// TwinCAT 3 PLC project PLC
// ProgramVersion: 3.1.4023.0
// libraries:
//   Tc2_Standard, * (Beckhoff Automation GmbH)
//   Tc2_System, * (Beckhoff Automation GmbH)
//   Tc2_Utilities, * (Beckhoff Automation GmbH)
//   Tc3_Module, * (Beckhoff Automation GmbH)
//   Util, * (System)
// project tree:
//   / PlcTask.TcTTO
//   POUs/ FB_ExportScopeData.TcPOU, FB_ScopeServerSample.TcPOU, MAIN.TcPOU
// real-time tasks:
//   TASK PlcTask: cycle T#10ms, priority 20, ADS port 350

CONFIGURATION PLC
    RESOURCE PLC ON TwinCAT3
        TASK PlcTask(INTERVAL := T#10ms, PRIORITY := 20);
        PROGRAM MAIN WITH PlcTask : MAIN;
    END_RESOURCE
END_CONFIGURATION

// ---- POUs/MAIN.TcPOU
PROGRAM MAIN
VAR
	fbBlink				:BLINK;
	Sinus				:GEN;
	SawTooth			:GEN;
	
	
	fbScopeServer		:FB_ScopeServerSample;
	
	xStartStopScope		:BOOL;
	xScopeBusy			:BOOL;
	xScopeError			:BOOL;
	iScopeErrorID		:UDINT;
	
	
	fbExportToCSV		:FB_ExportScopeData;
	xExport				:BOOL;
	xExportBusy			:BOOL;
	xExportError		:BOOL;
	iExportErrorID		:UDINT;
	
	
	//Example for listing files in a direcorty 
	//https://infosys.beckhoff.com/content/1033/tcplclib_tc2_utilities/35410571.html?id=3151343736833681439	
END_VAR

fbBlink(ENABLE:=TRUE , TIMELOW:=T#200MS , TIMEHIGH:=T#400MS);
Sinus(MODE:=GEN_MODE.SINUS , BASE:=TRUE , PERIOD:=T#1S , AMPLITUDE:=10000 );
SawTooth(MODE:=GEN_MODE.SAWTOOTH_RISE , BASE:=TRUE , PERIOD:=T#1S , AMPLITUDE:=10000 );



//Copy the "TemplateForPLC.tcscopex" file to the target system.
//TemplateForPLC.tcscopex file is a TwinCAT scope project.

fbScopeServer(
	sNetId					:='' , 
	bExternalTriggerEvent	:=xStartStopScope , 
	sConfigFile				:= 'C:\Scope\Templates\TemplateForPLC.tcscopex', 
	sSaveFile				:='C:\Scope\Records\Record1.svdx' , 
	bBusy					=>xScopeBusy , 
	bError					=>xScopeError, 
	nErrorId				=>iScopeErrorID);
	
	
//Copy the "ScopeExporterSettings.xml" file to the target system.
//ScopeExporterSettings.xml file was generated by using the scope export wizzard (Scope->Create Export Configuration)	
	
fbExportToCSV(
	sNetId					:='' , 
	bExport					:=xExport , 
	svd						:=fbScopeServer.sSaveFile , 
	target					:='C:\Scope\CSV\Record1.CSV' , 
	config					:='C:\Scope\Templates\ScopeExporterSettings.xml',
	bBusy					=>xExportBusy , 
	bError					=>xExportError , 
	iErrorID				=>iExportErrorID );

END_PROGRAM

// ---- POUs/FB_ScopeServerSample.TcPOU
FUNCTION_BLOCK FB_ScopeServerSample
VAR_INPUT
	sNetId					: STRING	:='';	
    bExternalTriggerEvent	: BOOL 		:= FALSE; //Rising edge start recording, falling edge stop and save
	sConfigFile				: STRING(80); //.tcscopex
	sSaveFile				: STRING(80); //.svdx
END_VAR
VAR_OUTPUT
    bBusy					: BOOL 		:= FALSE;
    bError					: BOOL 		:= FALSE;
    nErrorId				: UDINT 	:= 0;	
END_VAR
VAR

    bDone					: BOOL 		:= FALSE;	

    fbScopeServerControl	: FB_ScopeServerControl;
    eReqState				: E_ScopeServerState := SCOPE_SERVER_IDLE;
	
    eState					: (IDLE,RECORDING,SAVING,DISCONNECTING,ERROR,RESETING);
END_VAR

CASE eState OF
	IDLE:
		bBusy	:=FALSE;
		IF bExternalTriggerEvent THEN
			bBusy			:= TRUE;
	    	eReqState 		:= SCOPE_SERVER_START;
	    	eState 			:= RECORDING;	
		END_IF
	
	RECORDING:	
		IF fbScopeServerControl.bDone THEN
	    	IF NOT bExternalTriggerEvent THEN
	    	    eReqState 		:= SCOPE_SERVER_SAVE;
	    	    eState 			:= SAVING;
	    	END_IF
		ELSIF fbScopeServerControl.bError THEN
			eState	:=ERROR;		
		END_IF
		
	SAVING:
	    IF fbScopeServerControl.bDone THEN
	        eReqState 		:= SCOPE_SERVER_DISCONNECT;
			eState			:= DISCONNECTING;
		ELSIF fbScopeServerControl.bError THEN
			eState	:=ERROR;		
		END_IF
		
	DISCONNECTING:
		IF fbScopeServerControl.bDone THEN
	       eState := IDLE;
		ELSIF fbScopeServerControl.bError THEN
			eState	:=ERROR;				   
	    END_IF		
		
	ERROR:
		bBusy			:= FALSE;
		IF NOT bExternalTriggerEvent THEN
			bBusy			:= TRUE;
			eReqState 		:= SCOPE_SERVER_RESET;
			eState			:= DISCONNECTING;
		END_IF
		
	RESETING:
		IF fbScopeServerControl.bDone OR fbScopeServerControl.bError THEN
	       	eReqState 		:= SCOPE_SERVER_IDLE;
			eState			:= IDLE; 
	    END_IF		
		
END_CASE


fbScopeServerControl( sNetId		:= '',
                      eReqState		:= eReqState,
                      sConfigFile	:= sConfigFile,
                      sSaveFile		:= sSaveFile,
                      tTimeout		:= T#5S,
                      bBusy			=>,
                      bDone			=>bDone,
                      bError		=>bError,
                      nErrorId		=>nErrorId);

END_FUNCTION_BLOCK

// ---- POUs/FB_ExportScopeData.TcPOU
FUNCTION_BLOCK FB_ExportScopeData
VAR_INPUT
	sNetId			:STRING	:='';	
	bExport			:BOOL;
	svd 			:T_MaxString;//.svdx
	target			:T_MaxString;//.csv
	config			:T_MaxString;//.xml Configuration file created by export wizzard
	Channellist		:T_MaxString;//Channel List (Names of the channels(s) separated with semicolon
	start			:T_MaxString;//Starttime (As TwinCAT time stamp)
	end				:T_MaxString;//Endtime (As TwimCAT time stamp	
END_VAR
VAR_OUTPUT
	bBusy			:BOOL;
	bError			:BOOL;
	iErrorID		:UDINT;
END_VAR
VAR
	rtExport		:R_TRIG;
	fbStartExport	:NT_StartProcess;
	
	eState			:(IDEL,EXPORTING,ERROR);
	
    fbFormat   		: FB_FormatString2;
    sFormat    		: T_MaxString ;
	sCommand		: T_MaxString ;
END_VAR

rtExport(CLK:=bExport);
CASE eState OF 
	IDEL:
		bBusy		:=FALSE;
		IF rtExport.Q THEN
			bBusy		:=TRUE;
			//'"svd=c:\Scope Project.svdx" target=c:\TestExport.csv silent'
			sFormat:='"svd=%s" "target=%s"';
			
			IF config<>'' THEN
				sFormat:= CONCAT(sFormat,' "config=%s"');
			ELSE
				sFormat:= CONCAT(sFormat,'%s');
			END_IF

			IF Channellist<>'' THEN
				sFormat:= CONCAT(sFormat,' "Channellist=%s"');
			ELSE
				sFormat:= CONCAT(sFormat,'%s');
			END_IF
			
			IF start<>'' THEN
				sFormat:= CONCAT(sFormat,' "start=%s"');
			ELSE
				sFormat:= CONCAT(sFormat,'%s');
			END_IF			

			IF end<>'' THEN
				sFormat:= CONCAT(sFormat,' "end=%s"');
			ELSE
				sFormat:= CONCAT(sFormat,'%s');
			END_IF					
			
			sFormat	:= CONCAT(sFormat,' silent');
			
			fbFormat(
				pFormatString:=ADR(sFormat) , 
				arg1		:=F_STRING(svd) , 
				arg2		:=F_STRING(target) ,
				arg3		:=F_STRING(config), 
				arg4		:=F_STRING(Channellist), 
				arg5		:=F_STRING(start), 
				arg6		:=F_STRING(end), 				
				arg7		:=, 				
				pDstString	:=ADR(sCommand) , 
				nDstSize	:=SIZEOF(sCommand) );
				
			IF NOT fbFormat.bError THEN
				eState				:=EXPORTING;
				fbStartExport.START	:=TRUE;
			ELSE
				bError		:=fbFormat.bError;
				iErrorID	:=fbFormat.nErrId;
				eState		:=ERROR;
			END_IF
			
		END_IF
	
	EXPORTING:
		IF NOT fbStartExport.BUSY THEN
			fbStartExport.START	:=FALSE;
			IF NOT fbStartExport.ERR THEN
				eState		:=IDEL;
			ELSE
				bError		:=fbStartExport.ERR;
				iErrorID	:=fbStartExport.ERRID;
				eState		:=ERROR;				
			END_IF
		END_IF
	
	ERROR:
		eState		:=IDEL;
		
END_CASE


fbStartExport(
    NETID		:= sNetId, 
    PATHSTR		:= 'C:\TwinCAT\Functions\TE130X-Scope-View\TC3ScopeExportTool.exe', 
    DIRNAME		:= 'C:\TwinCAT\Functions\TE130X-Scope-View', 
    COMNDLINE	:= sCommand, 
    START		:= , 
    TMOUT		:= T#30S);

END_FUNCTION_BLOCK
